/// container for all communication data types that are used by the unit
TYPE XyTableComRef :
STRUCT
  Publish : REFERENCE TO XyTableComPublish; 
  Subscribe : REFERENCE TO XyTableComSubscribe; 
END_STRUCT
END_TYPE

(* stored: Version 1.1.0.1
   DUT XyTableComRef: Id {c856f270-fef8-4e0a-b1aa-aebfe63f2fd3} *)
